Staubli VAL3: english.pjx

Parameters version=s7.0 stackSize=5000 millimeterUnit=true
Program file=BuildTitle.pgx
Program file=Menu.pgx
Program file=Page.pgx
Program file=start.pgx
Program file=stop.pgx
Data file=english.dtx
Library alias=up path=Disk://Tracking/Tools/userPage/userPage.pjx
